// TIA Portal V18 export
// export: Created 2026-01-09T11:32:01.4763358Z, ExportSetting WithDefaults, DisplayName Totally Integrated Automation Portal, DisplayVersion V18 Update 5, DisplayName TIA Portal Openness, DisplayVersion V18 Update 5, DisplayName TIA Portal Teamcenter Gateway, DisplayVersion V18, DisplayName TIA Portal Version Control Interface, DisplayVersion V18, DisplayName SINAMICS Startdrive Advanced, DisplayVersion V18 SP2 Update 1, DisplayName SINAMICS Startdrive G110M, G120, G120C, G120D, G120P, G115D, DisplayVersion V18 SP2 Update 1, DisplayName SINAMICS Startdrive G130, G150, S120, S150, SINAMICS MV, S210, G220, S200, DisplayVersion V18 SP2 Update 1, DisplayName STEP 7 Professional, DisplayVersion V18 Update 5, DisplayName STEP 7 Safety, DisplayVersion V18, DisplayName WinCC Professional, DisplayVersion V18 Update 5
TagTable "Addon"
  Sys_VersionManagement_ProjectNumber : String  (PLC tag Sys.VersionManagement.ProjectNumber, CPU S71500-2PN_TP700, 1 s)
  Sys_VersionManagement_PLC IP Addr : Array [0..3] of UInt  (PLC tag Sys.VersionManagement."PLC IP Addr", CPU S71500-2PN_TP700, 1 s)
    TagArrayMember "[0]"
    TagArrayMember "[1]"
    TagArrayMember "[2]"
    TagArrayMember "[3]"
  Sys_VersionManagement_HMI IP Addr : Array [0..3] of UInt  (PLC tag Sys.VersionManagement."HMI IP Addr", CPU S71500-2PN_TP700, 1 s)
    TagArrayMember "[0]"
    TagArrayMember "[1]"
    TagArrayMember "[2]"
    TagArrayMember "[3]"
  Sys_VersionManagement_PLCVersion : Array [0..1] of UInt  (PLC tag Sys.VersionManagement.PLCVersion, CPU S71500-2PN_TP700, 1 s)
    TagArrayMember "[0]"
    TagArrayMember "[1]"
  Sys_VersionManagement_HMIVersion : Array [0..1] of UInt  (PLC tag Sys.VersionManagement.HMIVersion, CPU S71500-2PN_TP700, 1 s)
    TagArrayMember "[0]"
    TagArrayMember "[1]"
  Sys_VersionManagement_TIA Version : String  (PLC tag Sys.VersionManagement."TIA Version", CPU S71500-2PN_TP700, 1 s)
  Sys_VersionManagement_ProductLineName : String  (PLC tag Sys.VersionManagement.ProductLineName, CPU S71500-2PN_TP700, 1 s)
  Sys_VersionManagement_HMIPageID : Int  (PLC tag ST10_GeneralData.HMI.AREAPOINTER.SCREEN_NUMBER.SCREENNUMBER, CPU S71500-2PN_TP700, 1 s)
  Sys_VersionManagement_StationID : Int  (PLC tag Sys.VersionManagement.StationID, CPU S71500-2PN_TP700, 1 s)
